// TIA Portal V19 export
TYPE "LEXCHANGETRAY_typeSr1000ProfinetTelegram_errorStatusBits"
// stored: Access Published
   STRUCT
      statusByte : Byte;
      readFailure : Bool;
      presetFailure : Bool;
      registPresetFailure : Bool;
      tuneFailure : Bool;
      extReqFailure : Bool;
   END_STRUCT;
END_TYPE
